(* IEC 61131-3 sources: AXOpen/src/showcase/app/src/components.rexroth.press/Documentation, 2 files *)

(* ---- AxoSmartFunctionKit_v_4_x_x_Showcase.st ---- *)
USING AXOpen.Core;

NAMESPACE AXOpen.Components.Rexroth.Press.v_4_x_x

    {S7.extern=ReadWrite}
    CLASS AxoSmartFunctionKit_v_4_x_x_Showcase EXTENDS AXOpen.Core.AxoObject
        //<ComponentDeclaration>
        VAR PUBLIC
            AxoSmartFunctionKit : AXOpen.Components.Rexroth.Press.v_4_x_x.AxoSmartFunctionKit;
        END_VAR
        //</ComponentDeclaration>

        //<InitializationArgumentsDeclaration>
        VAR PUBLIC
            {#ix-set:AttributeName = "<#Activate manual control#>"}
            ActivateManualControl : BOOL;
        END_VAR
        //</InitializationArgumentsDeclaration>

        METHOD PUBLIC OVERRIDE Run
            VAR_INPUT
                inParent : IAxoObject;
            END_VAR

            SUPER.Run(inParent);

            IF ActivateManualControl THEN
                AxoSmartFunctionKit.ActivateManualControl();
            END_IF;

            //<Initialization>
            AxoSmartFunctionKit.Run(inParent              :=  THIS,
                                    hwID                :=  AXOpen.Showcase.HwIdentifiers#rexroth_press_HwID);

            AxoSmartFunctionKit.Config.InfoTime := T#10s;
            AxoSmartFunctionKit.Config.ErrorTime := T#30s;
            AxoSmartFunctionKit.Config.IpAddress := '192.168.100.240';
            AxoSmartFunctionKit.Config.CurveExportLocation := 'D:\Export';
            //</Initialization>

        THIS.UseInSequencer();
        END_METHOD

        //<Usage>
        VAR PUBLIC
            Sequencer : AxoSequencer;
            Steps : ARRAY[0..10] OF AXOpen.Core.AxoStep;
            {#ix-attr:[CompilerOmits()]}
            Request : AXOpen.Components.Rexroth.Press.v_4_x_x.AxoSmartFunctionKitRequest;
        END_VAR

        METHOD PRIVATE UseInSequencer

            Sequencer.Run(THIS);
            Sequencer.Open();
            Sequencer.SequenceMode:= eAxoSequenceMode#RunOnce;

            IF(Steps[0].Execute(Sequencer, 'SFK RESTORE')) THEN
                //-------------------------------------
                    ActivateManualControl := FALSE;
                    AxoSmartFunctionKit.Restore();
                    Sequencer.MoveNext();
                //-------------------------------------
            END_IF;

            IF(Steps[1].Execute(Sequencer, 'SFK RESET')) THEN
                //-------------------------------------
                    Request.Command := eAxoSmartFunctionKitCommand#ClearError;

                    IF AxoSmartFunctionKit.RunCommand(REF(Request)).IsDone() THEN
                        AxoSmartFunctionKit.Restore();
                        Sequencer.MoveNext();
                    END_IF;
                //-------------------------------------
            END_IF;

            IF(Steps[2].Execute(Sequencer, 'SFK STOP MOVEMENT')) THEN
                //-------------------------------------
                    Request.Command := eAxoSmartFunctionKitCommand#StopMovement;

                    IF AxoSmartFunctionKit.RunCommand(REF(Request)).IsDone() THEN
                        AxoSmartFunctionKit.Restore();
                        Sequencer.MoveNext();
                    END_IF;
                //-------------------------------------
            END_IF;

            IF(Steps[3].Execute(Sequencer, 'SFK HOME')) THEN
                //-------------------------------------
                    Request.Command := eAxoSmartFunctionKitCommand#StartHoming;

                    IF AxoSmartFunctionKit.RunCommand(REF(Request)).IsDone() THEN
                        AxoSmartFunctionKit.Restore();
                        Sequencer.MoveNext();
                    END_IF;
                //-------------------------------------
            END_IF;

            IF(Steps[4].Execute(Sequencer, 'SFK SET PROGRAM')) THEN
                //-------------------------------------
                    Request.Command     :=  eAxoSmartFunctionKitCommand#SetProgramActive;
                    Request.ProgramId   :=  2;

                    IF AxoSmartFunctionKit.RunCommand(REF(Request)).IsDone() THEN
                        AxoSmartFunctionKit.Restore();
                        Sequencer.MoveNext();
                    END_IF;
                //-------------------------------------
            END_IF;

            IF(Steps[5].Execute(Sequencer, 'SFK SET SERIAL ID')) THEN
                //-------------------------------------
                    Request.Command         :=  eAxoSmartFunctionKitCommand#StartProgram;
                    Request.SerialNumber    :=  System.Strings.Concat('Test_',System.Strings.ToString(THIS.GetContext().OpenCycleCount()));

                    Sequencer.MoveNext();
                //-------------------------------------
            END_IF;

            IF(Steps[6].Execute(Sequencer, 'SFK START PROGRAM')) THEN
                //-------------------------------------

                    IF AxoSmartFunctionKit.RunCommand(REF(Request)).IsDone() THEN
                        AxoSmartFunctionKit.Restore();
                        Sequencer.MoveNext();
                    END_IF;
                //-------------------------------------
            END_IF;

            IF(Steps[7].Execute(Sequencer, 'GET RESULTS')) THEN
                //-------------------------------------
                IF AxoSmartFunctionKit.GetResults().IsDone() THEN
                    AxoSmartFunctionKit.Restore();
                    Sequencer.MoveNext();
                END_IF;
                //-------------------------------------
            END_IF;

            IF(Steps[8].Execute(Sequencer, 'EXPORT CURVE')) THEN
                //-------------------------------------
                IF AxoSmartFunctionKit.ExportCurve().IsDone() THEN
                    AxoSmartFunctionKit.Restore();
                    Sequencer.MoveNext();
                END_IF;
                //-------------------------------------
            END_IF;

            IF(Steps[9].Execute(Sequencer, 'SEQUENCE DONE')) THEN
                //-------------------------------------
                Sequencer.CompleteSequence();
                //-------------------------------------
            END_IF;

        END_METHOD

        //</Usage>
    END_CLASS
END_NAMESPACE

(* ---- RexrothPress.st ---- *)
NAMESPACE AXOpen.Components.Rexroth.Press.v_4_x_x

    {S7.extern=ReadWrite}
    CLASS RexrothPress EXTENDS AXOpen.Core.AxoObject
        VAR PUBLIC
            _rootObject : AxoObject;
            axoSmartFunctionKit_v_4_x_x : AxoSmartFunctionKit_v_4_x_x_Showcase;
        END_VAR

        METHOD PUBLIC Execute
            _rootObject.Run(THIS);
            axoSmartFunctionKit_v_4_x_x.Run(_rootObject);
        END_METHOD
    END_CLASS
END_NAMESPACE
